PROGRAM P_MotionControl
VAR
	fbClock : FB_Clock;
	fTime : LREAL;
	bStartClock : BOOL;
	fbPrimaryControl : FB_ClosedLoopControl; 
	fPGain : LREAL := G_IO.P_Gain;//3.0;
	fIGain : LREAL := G_IO.I_Gain;//1.0;
	fbJoystick : FB_Joystick;
	fWinchVelRef : LREAL;
	fWinchPosRef : LREAL;
	fbWinchVelIntegrator : FB_Integrator;
	fbEncoder : FB_Encoder;
	fWinchPos : LREAL;
	fInitialWinchPos : LREAL;
	bWinchVelIntegratorOn: BOOL := TRUE; 
	fSineMotionGen : FB_SineMotionGenerator;
	PosRefTEST : LREAL; 
	bAutoEnable : BOOL;
	bManualEnable : BOOL;
	fSineDisplacementSp : LREAL := 0.3; // Nils Was here
	fSinePeriodeTime : LREAL := 5.0;
	fWinchPosRefManual : LREAL;
	// fWinchPosRefAuto : LREAL;  // THis is in the G_IO.fWinchPosRefAuto for HMI
	fbGetStartPos : FB_StartPos;
	fWinchVelRefManual : LREAL;
	fWinchVelRefAuto : LREAL;
	
	// Primary Control
	fWinchControlOutput : LREAL;
	fOutputPrimaryControl : LREAL;
	fInputSecondaryControl : LREAL := 1.0; 
	
	// Secoder control 
	fbSecondaryControl: FB_ClosedLoopControl;
	fOutputSecondaryControl : LREAL := 1.0;
	fSecondaryControlPGain : LREAL := 3.0; 
	fSecondaryControlIGain : LREAL := 1.0; 
	
 
	
	//Displacement Control
	fDisplacementNormalizedInput : LREAL := 1.0;
	fDisplacementInitial : LREAL := 1.0;
	fbDisplacementControl : FB_ClosedLoopControl;
	fDisplacementControlSignal : LREAL;
	fMaxDisplacement : LREAL := 1.0;
	fMinDisplacement : LREAL := 0.0;
	fbThDisplacement : FB_ThDisplacement;
	fThDisplacement_m3 : LREAL;
	fThDisplacement_cm3 : LREAL;
	fThDisplacement_norm : LREAL;
	
	/// Nils Was Here
	fDisplacementControldTryRef : LREAL; 
	fDisplacementControldLowring: LREAL; 
	fDisplacementControldHoysting: LREAL;
		
 	fDisplacementControldMinum: LREAL;
	fGOODHELPSIN : FB_SineMotionGenerator; 
	fSineDisplacementTest: LREAL; 
	fbTickTock : FB_Clock;
	 
	fSumControlerWithFilter : DisplacementSumWithFiller;
	
	
	fSeconderyPIDOut : LREAL; 
	
	//fWinchPosRefManualSC: LREAL;
	//fWinchVelRefManualSC: LREAL;   
	
	fbWinchVelIntegratorSC : FB_Integrator; 
	fbLogicBoxSC : FB_LogicBoxSC;
	
	fVelRefCos : LREAL; 
	ftestPostionrefSC: LREAL; 
	
	fbClosedLoopControlDC   : FB_ClosedLoopControlPID_DC; 
	fDisplacementControlPgainDC : LREAL := 2.0;
	fDisplacementControlIgainDC : LREAL := 2.0;
	fDisplacementControlDgainDC : LREAL := 2.0;
	fDerativeFilterCoeffientDC 	: LREAL := 100; 
 
	IntgrtorON : BOOL; 
	
	DomLineTest : LREAL; 
	fTestSignal : LREAL;
	fbLogicBoxSCz : FB_LogicBox2SC; 
	fTimeSC : LREAL; 
	
	fWinchPosRefSC : LREAL;
	
END_VAR
VAR // added by the converter: edge detectors and wires of the graphical bodies
    _w1 : INT;
    _w2, _w3 : BOOL;
END_VAR

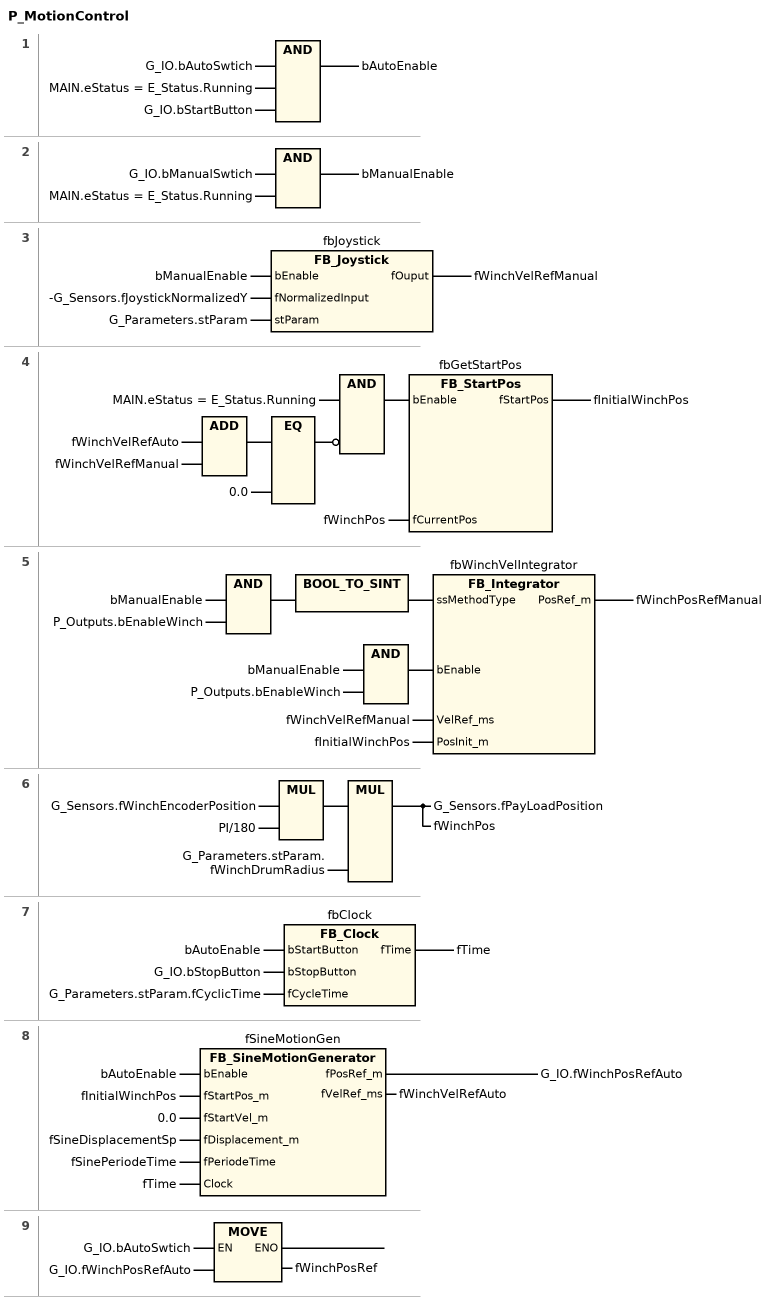
// NETWORK 1
bAutoEnable := G_IO.bAutoSwtich AND (MAIN.eStatus = E_Status.Running) AND G_IO.bStartButton;

// NETWORK 2
bManualEnable := G_IO.bManualSwtich AND (MAIN.eStatus = E_Status.Running);

// NETWORK 3
fbJoystick(
    bEnable := bManualEnable,
    fNormalizedInput := -G_Sensors.fJoystickNormalizedY,
    stParam := G_Parameters.stParam); // FB_Joystick
fWinchVelRefManual := fbJoystick.fOuput;

// NETWORK 4
fbGetStartPos(bEnable := (MAIN.eStatus = E_Status.Running) AND NOT (fWinchVelRefAuto + fWinchVelRefManual = 0.0), fCurrentPos := fWinchPos); // FB_StartPos
fInitialWinchPos := fbGetStartPos.fStartPos;

// NETWORK 5
fbWinchVelIntegrator(
    ssMethodType := BOOL_TO_SINT(bManualEnable AND P_Outputs.bEnableWinch),
    bEnable := bManualEnable AND P_Outputs.bEnableWinch,
    VelRef_ms := fWinchVelRefManual,
    PosInit_m := fInitialWinchPos); // FB_Integrator
fWinchPosRefManual := fbWinchVelIntegrator.PosRef_m;

// NETWORK 6
_w1 := (G_Sensors.fWinchEncoderPosition * (PI/180)) * G_Parameters.stParam.fWinchDrumRadius;
G_Sensors.fPayLoadPosition := _w1;
fWinchPos := _w1;

// NETWORK 7
fbClock(
    bStartButton := bAutoEnable,
    bStopButton := G_IO.bStopButton,
    fCycleTime := G_Parameters.stParam.fCyclicTime); // FB_Clock
fTime := fbClock.fTime;

// NETWORK 8
fSineMotionGen(
    bEnable := bAutoEnable,
    fStartPos_m := fInitialWinchPos,
    fStartVel_m := 0.0,
    fDisplacement_m := fSineDisplacementSp,
    fPeriodeTime := fSinePeriodeTime,
    Clock := fTime,
    fVelRef_ms => fWinchVelRefAuto); // FB_SineMotionGenerator
G_IO.fWinchPosRefAuto := fSineMotionGen.fPosRef_m;

// NETWORK 9
IF G_IO.bAutoSwtich THEN fWinchPosRef := G_IO.fWinchPosRefAuto; END_IF

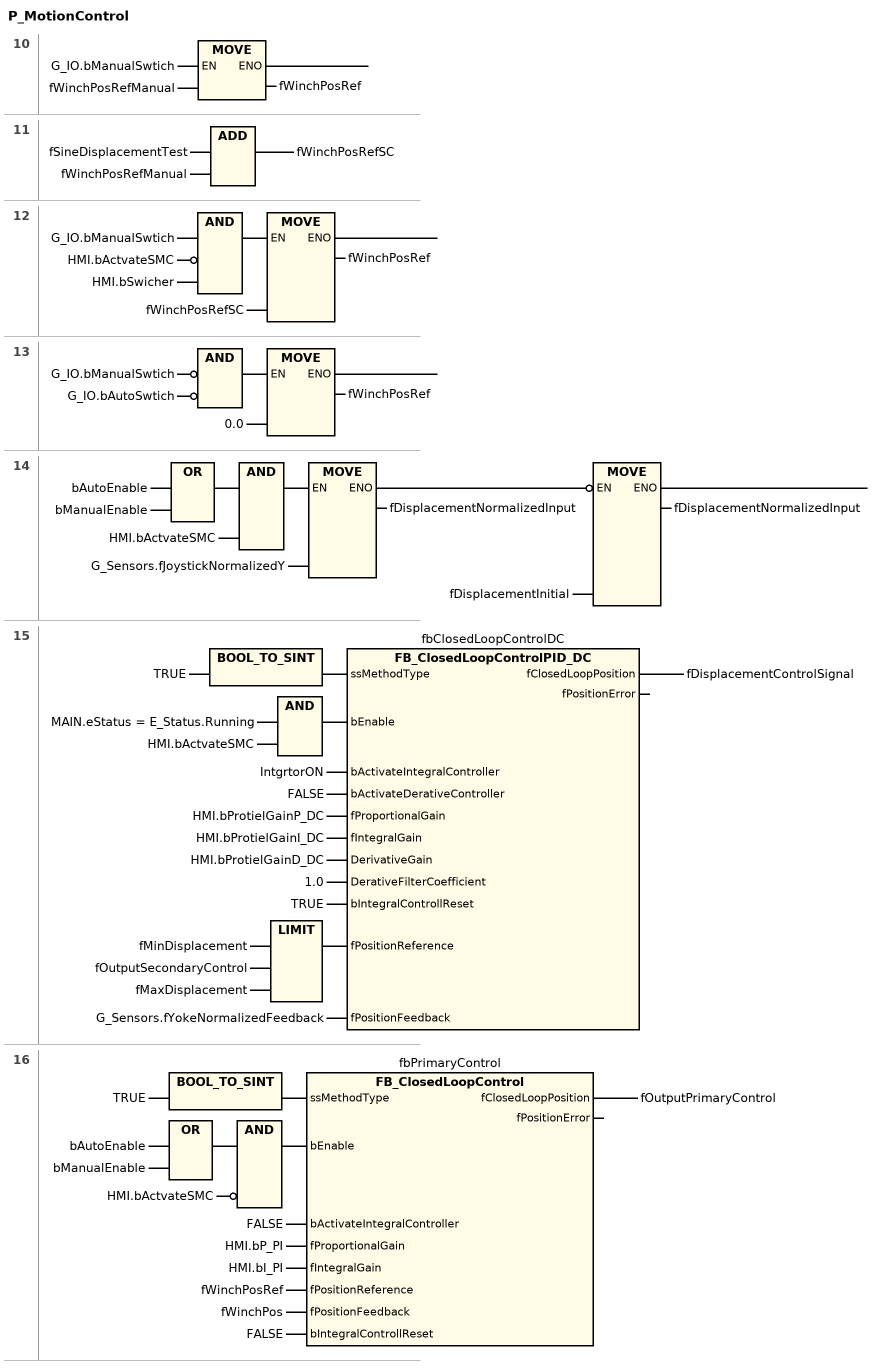
// NETWORK 10
IF G_IO.bManualSwtich THEN fWinchPosRef := fWinchPosRefManual; END_IF

// NETWORK 11
fWinchPosRefSC := fSineDisplacementTest + fWinchPosRefManual;

// NETWORK 12
IF G_IO.bManualSwtich AND NOT HMI.bActvateSMC AND HMI.bSwicher THEN fWinchPosRef := fWinchPosRefSC; END_IF

// NETWORK 13
IF NOT G_IO.bManualSwtich AND NOT G_IO.bAutoSwtich THEN fWinchPosRef := 0.0; END_IF

// NETWORK 14
_w2 := (bAutoEnable OR bManualEnable) AND HMI.bActvateSMC;
IF _w2 THEN fDisplacementNormalizedInput := G_Sensors.fJoystickNormalizedY; END_IF
IF NOT _w2 THEN fDisplacementNormalizedInput := fDisplacementInitial; END_IF

// NETWORK 15
fbClosedLoopControlDC(
    ssMethodType := BOOL_TO_SINT(TRUE),
    bEnable := (MAIN.eStatus = E_Status.Running) AND HMI.bActvateSMC,
    bActivateIntegralController := IntgrtorON,
    bActivateDerativeController := FALSE,
    fProportionalGain := HMI.bProtielGainP_DC,
    fIntegralGain := HMI.bProtielGainI_DC,
    DerivativeGain := HMI.bProtielGainD_DC,
    DerativeFilterCoefficient := 1.0,
    bIntegralControllReset := TRUE,
    fPositionReference := LIMIT(fMinDisplacement, fOutputSecondaryControl, fMaxDisplacement),
    fPositionFeedback := G_Sensors.fYokeNormalizedFeedback); // FB_ClosedLoopControlPID_DC
fDisplacementControlSignal := fbClosedLoopControlDC.fClosedLoopPosition;

// NETWORK 16
fbPrimaryControl(
    ssMethodType := BOOL_TO_SINT(TRUE),
    bEnable := (bAutoEnable OR bManualEnable) AND NOT HMI.bActvateSMC,
    bActivateIntegralController := FALSE,
    fProportionalGain := HMI.bP_PI,
    fIntegralGain := HMI.bI_PI,
    fPositionReference := fWinchPosRef,
    fPositionFeedback := fWinchPos,
    bIntegralControllReset := FALSE); // FB_ClosedLoopControl
fOutputPrimaryControl := fbPrimaryControl.fClosedLoopPosition;

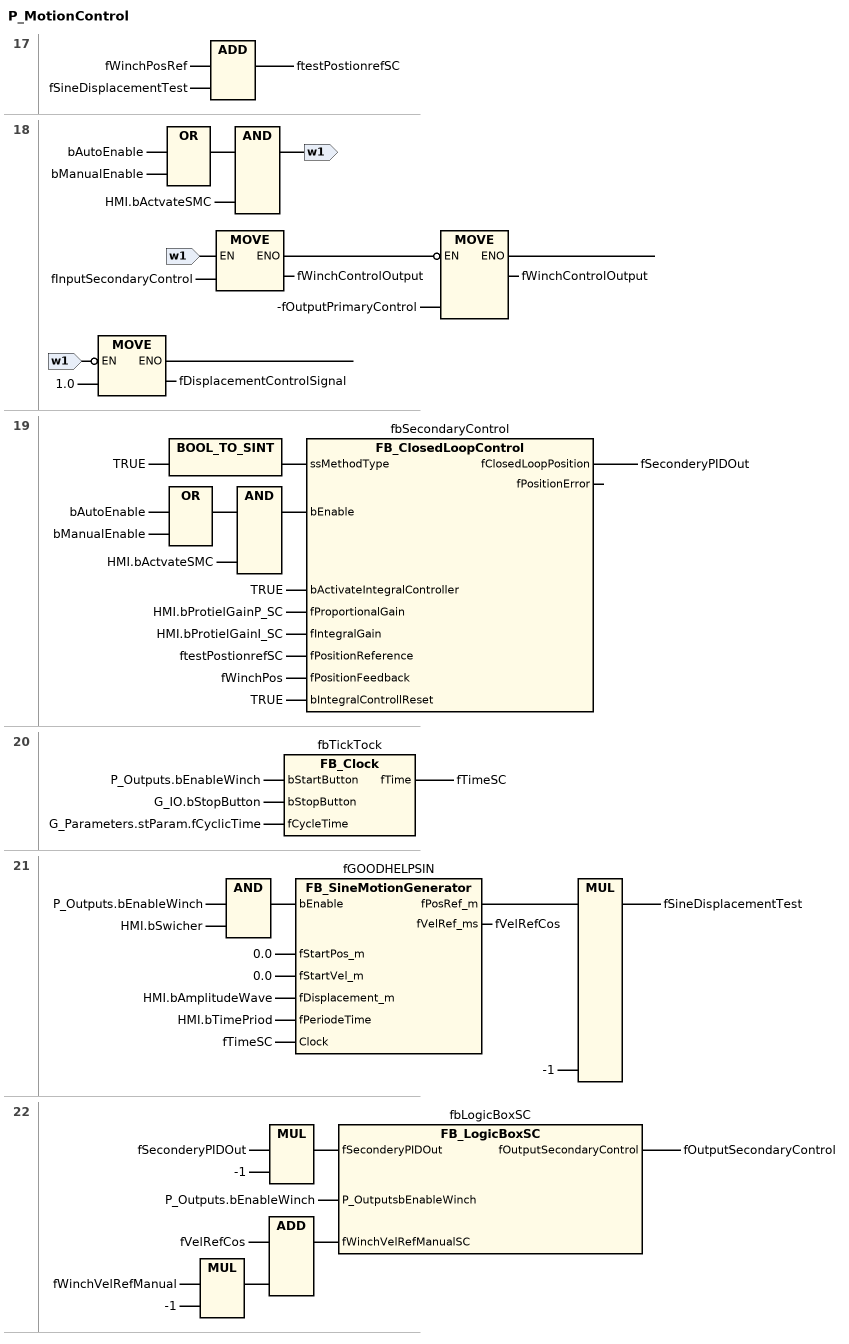
// NETWORK 17
ftestPostionrefSC := fWinchPosRef + fSineDisplacementTest;

// NETWORK 18
_w3 := (bAutoEnable OR bManualEnable) AND HMI.bActvateSMC;
IF _w3 THEN fWinchControlOutput := fInputSecondaryControl; END_IF
IF NOT _w3 THEN fWinchControlOutput := -fOutputPrimaryControl; END_IF
IF NOT _w3 THEN fDisplacementControlSignal := 1.0; END_IF

// NETWORK 19
fbSecondaryControl(
    ssMethodType := BOOL_TO_SINT(TRUE),
    bEnable := (bAutoEnable OR bManualEnable) AND HMI.bActvateSMC,
    bActivateIntegralController := TRUE,
    fProportionalGain := HMI.bProtielGainP_SC,
    fIntegralGain := HMI.bProtielGainI_SC,
    fPositionReference := ftestPostionrefSC,
    fPositionFeedback := fWinchPos,
    bIntegralControllReset := TRUE); // FB_ClosedLoopControl
fSeconderyPIDOut := fbSecondaryControl.fClosedLoopPosition;

// NETWORK 20
fbTickTock(
    bStartButton := P_Outputs.bEnableWinch,
    bStopButton := G_IO.bStopButton,
    fCycleTime := G_Parameters.stParam.fCyclicTime); // FB_Clock
fTimeSC := fbTickTock.fTime;

// NETWORK 21
fGOODHELPSIN(
    bEnable := P_Outputs.bEnableWinch AND HMI.bSwicher,
    fStartPos_m := 0.0,
    fStartVel_m := 0.0,
    fDisplacement_m := HMI.bAmplitudeWave,
    fPeriodeTime := HMI.bTimePriod,
    Clock := fTimeSC,
    fVelRef_ms => fVelRefCos); // FB_SineMotionGenerator
fSineDisplacementTest := fGOODHELPSIN.fPosRef_m * -1;

// NETWORK 22
fbLogicBoxSC(
    fSeconderyPIDOut := fSeconderyPIDOut * -1,
    P_OutputsbEnableWinch := P_Outputs.bEnableWinch,
    fWinchVelRefManualSC := fVelRefCos + fWinchVelRefManual * -1); // FB_LogicBoxSC
fOutputSecondaryControl := fbLogicBoxSC.fOutputSecondaryControl;

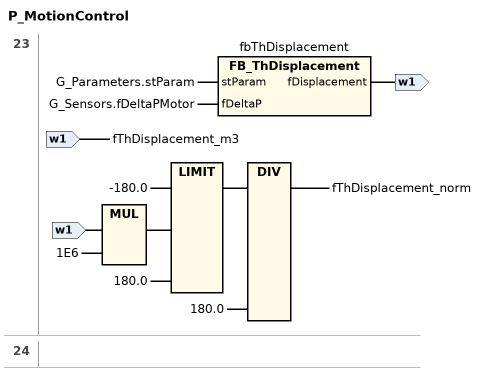
// NETWORK 23
fbThDisplacement(stParam := G_Parameters.stParam, fDeltaP := G_Sensors.fDeltaPMotor); // FB_ThDisplacement
fThDisplacement_m3 := fbThDisplacement.fDisplacement;
fThDisplacement_norm := LIMIT(-180.0, fbThDisplacement.fDisplacement * 1E6, 180.0) / 180.0;

// NETWORK 24

END_PROGRAM

(* stored: Version 1.1.0.1, ProductVersion 3.1.4024.12
   POU P_MotionControl: Id {fca9df39-4db4-416e-89b5-b1157c751beb}, SpecialFunc None *)
